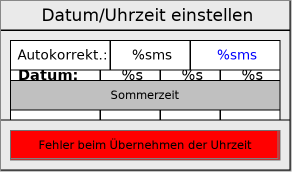
VISUALIZATION V_SetTime  // 292x172
VAR_IN_OUT
  IOfbSystemCX : FB_SystemCX;
END_VAR
    Rectangle (0,30 290x140), "Achtung: Es wird die Winterzeit eingestellt!", invisible if: IOfbSystemCX.VbSetTimeStart = 0
    Rectangle (0,30 290x90), invisible if: IOfbSystemCX.VbSetTimeStart = 1
    Rectangle (0,0 290x30), "Datum/Uhrzeit einstellen", colour toggle: IOfbSystemCX.VbSetTimeStart
        toggle IOfbSystemCX.VbSetTimeStart
    Rectangle (220,60 60x30), "%s", text variable: IOfbSystemCX.INstSysTimeDate.wDay, invisible if: IOfbSystemCX.VbSetTimeStart = 0
        OnMouseDown: write the text variable via Edit, min 1, max 31
    Rectangle (10,60 90x30), "Datum:", invisible if: IOfbSystemCX.VbSetTimeStart = 0
    Rectangle (10,90 90x30), "Uhrzeit:", invisible if: IOfbSystemCX.VbSetTimeStart = 0
    Rectangle (160,60 60x30), "%s", text variable: IOfbSystemCX.INstSysTimeDate.wMonth, invisible if: IOfbSystemCX.VbSetTimeStart = 0
        OnMouseDown: write the text variable via Edit, min 1, max 12
    Rectangle (100,60 60x30), "%s", text variable: IOfbSystemCX.INstSysTimeDate.wYear, invisible if: IOfbSystemCX.VbSetTimeStart = 0
        OnMouseDown: write the text variable via Edit, min 2016, max 2099
    Rectangle (100,90 60x30), "%s", text variable: IOfbSystemCX.INstSysTimeDate.wHour, invisible if: IOfbSystemCX.VbSetTimeStart = 0
        OnMouseDown: write the text variable via Edit, min 0, max 23
    Rectangle (160,90 60x30), "%s", text variable: IOfbSystemCX.INstSysTimeDate.wMinute, invisible if: IOfbSystemCX.VbSetTimeStart = 0
        OnMouseDown: write the text variable via Edit, min 0, max 59
    Rectangle (220,90 60x30), "%s", text variable: IOfbSystemCX.INstSysTimeDate.wSecond, invisible if: IOfbSystemCX.VbSetTimeStart = 0
        OnMouseDown: write the text variable via Edit, min 0, max 59
    Rectangle (10,40 100x30), "Autokorrekt.:", tooltip "Automatische Korrektur der Uhrzeit je Tag", invisible if: IOfbSystemCX.VbSetTimeStart = 1
    Rectangle (110,40 80x30), "%sms", tooltip "Automatische Korrektur der Uhrzeit je Tag", text variable: IOfbSystemCX.VnviTimeCorrectionEachDay, invisible if: IOfbSystemCX.VbSetTimeStart = 1
        OnMouseDown: write the text variable via Default, min -10000, max 10000
    Rectangle (190,40 90x30), "%sms", tooltip "aktueller Korrekturwert", text variable: IOfbSystemCX.nviTimeCorrectionSum, invisible if: IOfbSystemCX.VbSetTimeStart = 1
        OnMouseDown: write the text variable via Default, min -99999, max 99999
    Button (10,130 130x30), "Abbrechen", invisible if: IOfbSystemCX.VbSetTimeStart = 0
        tap PLC_PRG.bSetClock
        toggle IOfbSystemCX.VbSetTimeStart
    Button (140,130 140x30), "Übernehmen", invisible if: IOfbSystemCX.VbSetTimeStart = 0
        tap PLC_PRG.bSetClock
        toggle IOfbSystemCX.VbSetTimeReturn
    Button (10,130 270x30), "Fehler beim Übernehmen der Uhrzeit", invisible if: IOfbSystemCX.VbSetTimeError = 0
        tap PLC_PRG.bSetClock
        toggle IOfbSystemCX.VbSetTimeStart
    Rectangle (10,80 270x30), "Sommerzeit", colour toggle: IOfbSystemCX.nvbSummerTime, invisible if: IOfbSystemCX.VbSetTimeStart = 1
        toggle IOfbSystemCX.nvbSummerTime
END_VISUALIZATION

(* stored: Version 1.1.0.1, ProductVersion 3.1.4018.9
   Visu V_SetTime: Id {a1654042-ff52-4b1a-a8cf-5bed84732d1f} *)
